(* IEC 61131-3 sources: Std_PalletMover/Class/FunctionBase, 1 file *)

(* ---- FunctionBase.st ---- *)
(*!
<Class
	Name               = "FunctionBase"
	Revision           = "0.0"
	RealtimeTask       = "false"
	CyclicTask         = "false"
	BackgroundTask     = "false"
	Sigmatek           = "false"
	OSInterface        = "false"
	HighPriority       = "false"
	Automatic          = "false"
	UpdateMode         = "Prescan"
	SharedCommandTable = "true"
	Objectsize         = "(570,120)">
	<Channels>
	</Channels>
	<Network Name="FunctionBase">
		<!-- List of Components in this network -->
		<Components>
			<Object
				Name       = "_base"
				Class      = "LinkedObjectBase"
				Position   = "(218,120)"
				Visualized = "false">
				<Channels>
					<Server Name="ObjectStatus"/>
					<Server Name="ToObject"/>
					<Client Name="op_LogData"/>
					<Client Name="p_NextObject"/>
					<Client Name="p_PreviousObject"/>
				</Channels>
			</Object>
		</Components>
		<Comments>
		</Comments>
		<!-- List of Connections in this network -->
		<Connections>
			<Connection Source="this.ToObject" Destination="_base.ToObject" Vertices="(1060,210),(888,210),"/>
			<Connection Source="_base.p_NextObject" Destination="this.p_NextObject" Vertices="(218,330),(38,270),"/>
			<Connection Source="_base.op_LogData" Destination="this.op_LogData" Vertices="(218,210),(38,210),"/>
			<Connection Source="this.ObjectStatus" Destination="_base.ObjectStatus" Vertices="(1060,270),(888,270),"/>
		</Connections>
		<!-- Headerfiles -->
		<Options>
		</Options>
	</Network>
</Class>
*)
#pragma using LinkedObjectBase

FunctionBase : CLASS
: LinkedObjectBase
	TYPE
	  PeripheralStatus : BDINT
	  [
	    1 ConfigurationReady,
	    2 Startupready,
	    3 StetingsLoaded,
	    4 Operational,
	    5 Bit5,
	    6 Bit6,
	    7 Bit7,
	    8 Bit8,
	    9 Bit9,
	    10 Bit10,
	    11 Bit11,
	    12 Bit12,
	    13 Bit13,
	    14 Bit14,
	    15 Bit15,
	    16 Bit16,
	    17 Bit17,
	    18 Bit18,
	    19 Bit19,
	    20 Bit20,
	    21 Bit21,
	    22 Bit22,
	    23 Bit23,
	    24 Bit24,
	    25 Bit25,
	    26 Bit26,
	    27 Bit27,
	    28 Bit28,
	    29 Bit29,
	    30 Bit30,
	    31 Bit31,
	    32 InError,
	  ];
	END_TYPE
  //Servers:
  //Clients:
  //Variables:
  //Functions:

	FUNCTION VIRTUAL GLOBAL HandleOperational
		VAR_OUTPUT
			RetValue 	: DINT;
		END_VAR;

	FUNCTION VIRTUAL GLOBAL Handleconfiguration
		VAR_OUTPUT
			RetValue 	: DINT;
		END_VAR;

	FUNCTION VIRTUAL GLOBAL HandleGetSettings
		VAR_OUTPUT
			RetValue 	: DINT;
		END_VAR;

	FUNCTION VIRTUAL GLOBAL HandleStartUp
		VAR_OUTPUT
			RetValue 	: DINT;
		END_VAR;
  //Tables:
	FUNCTION @STD
		VAR_OUTPUT
			ret_code	: CONFSTATES;
		END_VAR;
	FUNCTION GLOBAL TAB @CT_;
END_CLASS;

FUNCTION VIRTUAL GLOBAL FunctionBase::HandleOperational
	VAR_OUTPUT
		RetValue 	: DINT;
	END_VAR

END_FUNCTION

FUNCTION VIRTUAL GLOBAL FunctionBase::Handleconfiguration
	VAR_OUTPUT
		RetValue 	: DINT;
	END_VAR

END_FUNCTION

FUNCTION VIRTUAL GLOBAL FunctionBase::HandleGetSettings
	VAR_OUTPUT
		RetValue 	: DINT;
	END_VAR

END_FUNCTION

FUNCTION VIRTUAL GLOBAL FunctionBase::HandleStartUp
	VAR_OUTPUT
		RetValue 	: DINT;
	END_VAR

END_FUNCTION
